FUNCTION_BLOCK DeserializationErrorFactory_TestSuite EXTENDS TcUnit.FB_TestSuite

TestCreateICustomDeserializationFailedError();
TestCreateIncorrectKeyTypeError();
TestCreateIncorrectTypeError();
TestCreateMissingKeyError();
TestCreateInvalidKeyError();

METHOD PUBLIC TestCreateICustomDeserializationFailedError
VAR
	error : CustomDeserializationFailedError('testMessage');
	factory : DeserializationErrorFactory;
	newError : I_Error;
END_VAR
TEST('TestCreateICustomDeserializationFailedError');

newError := factory.CreateCustomDeserializationFailedError('testMessage');

AssertTrue(
	Condition := newError.IsSameAs(error),
	Message := 'Did not produce the correct error type'
);

AssertEquals_String(
	Actual := newError.Message,
	Expected := error.Message,
	Message := 'Did not produce error with correct message'
);

newError.Dispose();

TEST_FINISHED();
END_METHOD

METHOD PUBLIC TestCreateIncorrectKeyTypeError
VAR
	error : IncorrectKeyTypeDeserializationError('testType', 'testKey');
	factory : DeserializationErrorFactory;
	newError : I_Error;
END_VAR
TEST('TestCreateIncorrectKeyTypeError');

newError := factory.CreateIncorrectKeyTypeError('testType','testKey');

AssertTrue(
	Condition := newError.IsSameAs(error),
	Message := 'Did not produce the correct error type'
);

AssertEquals_String(
	Actual := newError.Message,
	Expected := error.Message,
	Message := 'Did not produce error with correct message'
);

newError.Dispose();

TEST_FINISHED();
END_METHOD

METHOD PUBLIC TestCreateIncorrectTypeError
VAR
	error : IncorrectTypeDeserializationError('testType');
	factory : DeserializationErrorFactory;
	newError : I_Error;
END_VAR
TEST('TestCreateIncorrectTypeError');

newError := factory.CreateIncorrectTypeError('testType');

AssertTrue(
	Condition := newError.IsSameAs(error),
	Message := 'Did not produce the correct error type'
);

AssertEquals_String(
	Actual := newError.Message,
	Expected := error.Message,
	Message := 'Did not produce error with correct message'
);

newError.Dispose();

TEST_FINISHED();
END_METHOD

METHOD PUBLIC TestCreateInvalidKeyError
VAR
	error : InvalidKeyDeserializationError;
	factory : DeserializationErrorFactory;
	newError : I_Error;
END_VAR
TEST('TestCreateInvalidKeyError');

newError := factory.CreateInvalidKeyError();

AssertTrue(
	Condition := newError.IsSameAs(error),
	Message := 'Did not produce the correct error type'
);

AssertEquals_String(
	Actual := newError.Message,
	Expected := error.Message,
	Message := 'Did not produce error with correct message'
);

newError.Dispose();

TEST_FINISHED();
END_METHOD

METHOD PUBLIC TestCreateMissingKeyError
VAR
	error : MissingKeyDeserializationError('testKey');
	factory : DeserializationErrorFactory;
	newError : I_Error;
END_VAR
TEST('TestCreateMissingKeyError');

newError := factory.CreateMissingKeyError('testKey');

AssertTrue(
	Condition := newError.IsSameAs(error),
	Message := 'Did not produce the correct error type'
);

AssertEquals_String(
	Actual := newError.Message,
	Expected := error.Message,
	Message := 'Did not produce error with correct message'
);

newError.Dispose();

TEST_FINISHED();
END_METHOD

END_FUNCTION_BLOCK

(* stored: Version 1.1.0.1, ProductVersion 3.1.4024.12
   POU DeserializationErrorFactory_TestSuite: Id {7b79ae16-928f-4457-901a-acc38e140e45}, SpecialFunc None
   Method TestCreateICustomDeserializationFailedError: Id {d1bb8acc-7f87-0a23-05ce-525a905e0def}
   Method TestCreateIncorrectKeyTypeError: Id {aadd7fdd-882e-4d73-b70b-a590bfe89472}
   Method TestCreateIncorrectTypeError: Id {1926c914-755f-4a3f-a386-540e03b20ba0}
   Method TestCreateInvalidKeyError: Id {10e57135-1740-4d69-8446-48b2c211a9cf}
   Method TestCreateMissingKeyError: Id {cf5ec45e-2a5d-4a07-b6d3-fbbe9e9b4b39} *)
